ABB RobotStudio station: Solution 4 with position track.rspag

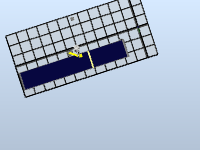
--- station ---
Station Solution4 (saved by RobotStudio 6.8.8148.134)
Controller System1, task T_ROB1: task frame (RAPID world) sits at (5535.63, 748.67, 709.58) mm in the station
Controller System1
  mechanical unit ROB_1: IRB1600_10_145__01, 6 joints, base frame (480.91, -513.23, -359.58) mm, rotated rx 0 ry 0 rz 90 deg
  mechanical unit CNV1: ?, 1 joints, base frame (0, 0, 0) mm
Layout (positions relative to the parent item):
  - bin mover_3 [smart component, from libraries\bin mover.rslib] at (-500, 0, 0) mm
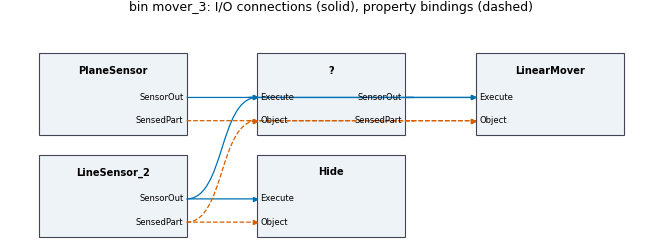
      connections:
        ?.SensorOut -> LinearMover.Execute
        PlaneSensor.SensorOut -> LinearMover.Execute
        ?.SensorOut -> ?.Execute
        LineSensor_2.SensorOut -> ?.Execute
        LineSensor_2.SensorOut -> Hide.Execute
        ?.SensedPart => LinearMover.Object
        PlaneSensor.SensedPart => LinearMover.Object
        ?.SensedPart => ?.Object
        LineSensor_2.SensedPart => ?.Object
        LineSensor_2.SensedPart => Hide.Object
    - LinearMover [smart component, from Components\LinearMover.rslib] at (6663.26, 677.27, 1050.93) mm, rotated rx 180 ry 0 rz 90 deg
        properties: Object=(none); Direction=[0 0 -1]; Speed=8; Reference=Global; ReferenceObject=(none)
    - PlaneSensor [smart component, from Components\PlaneSensor.rslib]
        properties: Origin=[7.419145 0.146999 1.42]; Axis1=[0 0 -1.35]; Axis2=[0 0.4 0]; SensedPart=(none)
      - _sensorPart_ [part, from libraries\bin mover.rslib]
    - LineSensor_2 [smart component, from Components\LineSensor.rslib]
        properties: Start=[7.369145 0.346999 0.008]; End=[7.369145 0.346999 0.123]; Radius=0.09; SensedPart=(none); SensedPoint=[0 0 0]
      - _sensorPart_ [part, from libraries\bin mover.rslib]
    - Hide [smart component, from Components\Hide.rslib]
        properties: Object=(none)
  - bin1_2 [part, from libraries\bin1.rslib] at (6733.74, 347, -12) mm
  - conveyor 1 [part] at (0, -1500, -4460) mm, rotated rx 90 ry 0 rz 90 deg
  - Suction gripper 18cm [smart component] at (6041.96, 965.18, 1386.5) mm, rotated rx 180 ry 0 rz -90 deg
      signals: DI do1
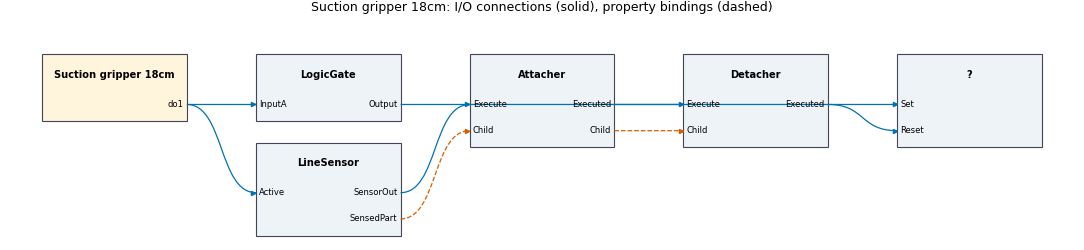
      connections:
        Suction gripper 18cm.do1 -> LogicGate.InputA
        Suction gripper 18cm.do1 -> LineSensor.Active
        LogicGate.Output -> Detacher.Execute
        LineSensor.SensorOut -> Attacher.Execute
        Attacher.Executed -> ?.Set
        Detacher.Executed -> ?.Reset
        LineSensor.SensedPart => Attacher.Child
        Attacher.Child => Detacher.Child
    - Attacher [smart component, from Components\Attacher.rslib]
        properties: Parent=Suction_gripper 18cm; Flange=0; Child=Yellow block; Mount=false; Offset=[0 0 0]; Orientation=[0 0 0]
    - LogicGate [smart component, from Components\LogicGate.rslib]
        properties: Operator=NOT; Delay=0
    - LineSensor [smart component, from Components\LineSensor.rslib] at (7150.29, 306.47, 1168.39) mm, rotated rx 180 ry 0 rz 90 deg
        properties: Start=[-0.30577796087058 -7.14894421240012 1.16938863540814]; End=[-0.305777964813962 -7.14894420825673 1.13938863540814]; Radius=0.09; SensedPart=Yellow block; SensedPoint=[6.72294091796875 0.422247802734375 1.36320727539063]
      - _sensorPart_ [part]
    - Detacher [smart component, from Components\Detacher.rslib]
        properties: Child=Yellow block; KeepPosition=true
  - Suction_gripper 18cm [mechanism, from libraries\Suction_gripper_18cm.rslib] at (6041.96, 965.18, 1471.5) mm, rotated rx 180 ry 0 rz -90 deg
  - IRB1600_10_145__01 [mechanism, from Robots\IRB1600_10_145_G_01.rslib] at (6016.55, 235.44, 350) mm, rotated rx 0 ry 0 rz 90 deg; joint values [-0.0348, -0.0283, 0.0278, 0, 1.5713, -0.0348] (rad or m)
  - 输送链 [conveyor]
    - Conveyor cover [part] at (-300, 0, 14) mm
    - Yellow block [part] at (0, -475.41, 0) mm
    - 传送带对象_37 [conveyorobject] at (9300.11, 748.67, 709.58) mm
      - Yellow block [part] at (-383.96, -1767.23, -1501.67) mm
    - 传送带对象_38 [conveyorobject] at (6600.11, 748.67, 709.58) mm
      - Yellow block [part] at (-344.85, -1769.56, -1503.25) mm
    - 传送带对象_39 [conveyorobject] at (3900.11, 748.67, 709.58) mm
      - Yellow block [part] at (-1067.12, -1221.88, -152.65) mm
  - SmartComponent_1 [smart component]
      signals: DI do_rapid
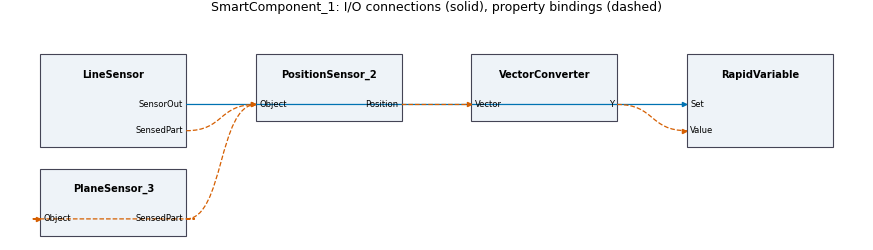
      connections:
        LineSensor.SensorOut -> RapidVariable.Set
        PlaneSensor_3.SensedPart => LinearMover.Object
        PlaneSensor_3.SensedPart => PositionSensor_2.Object
        LineSensor.SensedPart => PositionSensor_2.Object
        PositionSensor_2.Position => VectorConverter.Vector
        VectorConverter.Y => RapidVariable.Value
    - RapidVariable [smart component, from Components\RapidVariable.rslib]
        properties: DataType=num; Controller=System1; Task=T_ROB1; Module=Module1; Variable=y; Value=0.20905832662045
    - PositionSensor_2 [smart component, from Components\PositionSensor.rslib]
        properties: Object=(none); Reference=Object; ReferenceObject=Reference; Position=[-0.750554000259359 0.20905832662045 -0.741395]; Orientation=[0 0 0]
    - LineSensor [smart component, from Components\LineSensor.rslib]
        properties: Start=[5.101063 2.339147 0.72958]; End=[5.101063 0.739147 0.72958]; Radius=0.02; SensedPart=(none); SensedPoint=[0 0 0]
      - _sensorPart_ [part]
    - VectorConverter [smart component, from Components\VectorConverter.rslib]
        properties: X=-0.750554000259359; Y=0.20905832662045; Z=-0.741395; Vector=[-0.750554000259359 0.20905832662045 -0.741395]
  - Reference [part] at (3022.67, -345.33, 752.97) mm
  - Random position [smart component]
      connections:
        PlaneSensor.SensorOut -> Random.Execute
        PlaneSensor.SensorOut -> LinearMover.Execute
        PlaneSensor.SensedPart => LinearMover.Object
        Random.Value => LinearMover.Speed
    - Random [smart component, from Components\Random.rslib]
        properties: Value=0.673263867373236; Min=-0.1; Max=1.2
    - PlaneSensor [smart component, from Components\PlaneSensor.rslib]
        properties: Origin=[4.525795 0.752121 0.710084]; Axis1=[0 0 0.18]; Axis2=[0 1.575 0]; SensedPart=(none)
      - _sensorPart_ [part]
    - LinearMover [smart component, from Components\LinearMover.rslib]
        properties: Object=(none); Direction=[0 0.001 0]; Speed=0.673263867373236; Reference=Global; ReferenceObject=(none)
Attachment: Suction gripper 18cm is attached to Suction_gripper 18cm / Suction gripper 18cm
Attachment: Suction_gripper 18cm is attached to IRB1600_10_145__01 / Link6
Conveyor tracking 连接_2: unit CNV1, TravelOffset=3.7, QueueTrackDistance=0, StartWindowWidth=1.8, SyncSeparation=0, CountsPerMeter=10000
Station logic (signal -> signal, property => property):
  System1.do_attach -> Suction gripper 18cm.do1

--- Backups/System1/RAPID/TASK1/PROGMOD/CalibData.mod ---
MODULE CalibData
	TASK PERS wobjdata wobj_cnv1:=[FALSE,FALSE,"CNV1",[[0,0,0],[1,0,0,0]],[[0,0,0],[1,0,0,0]]];
ENDMODULE

--- Backups/System1/RAPID/TASK1/PROGMOD/Module1.mod ---
MODULE Module1
    VAR num y:=0;
	CONST robtarget Target_10:=[[480.915,236.77,676.92],[0,-0.707106781,0.707106781,0],[0,0,0,0],[9E+09,9E+09,9E+09,9E+09,9E+09,0]];
	CONST robtarget Target_20:=[[29.699626144,355.874016057,111.58001204],[0.000000002,0.707106781,-0.707106781,0.000000007],[0,-1,0,0],[9E+09,9E+09,9E+09,9E+09,9E+09,0]];
	CONST robtarget Target_30:=[[1192.207950487,-330.312717415,676.919992598],[0.000000021,0.707106781,-0.707106781,0.000000022],[-1,-1,-1,0],[9E+09,9E+09,9E+09,9E+09,9E+09,0]];
    PERS tooldata Suction_gripper_18cm:=[TRUE,[[0,0,85],[1,0,0,0]],[1,[0,0,1],[1,0,0,0],0,0,0]];

    PROC main()
        ActUnit CNV1;

        WHILE 2>1 DO

            WaitWObj wobj_cnv1;
            Path_10;
            DropWObj wobj_cnv1;

        ENDWHILE
    ENDPROC
    PROC Path_10()
		MoveL Target_10,vmax,fine,Suction_gripper_18cm\WObj:=wobj0;
		MoveL reltool(Target_20,-y*1000,0,0),vmax,z10,Suction_gripper_18cm\WObj:=wobj_cnv1;
		Set do_attach;
		MoveL Target_30,vmax,fine,Suction_gripper_18cm\WObj:=wobj0;
		Reset do_attach;
		MoveL Target_10,vmax,fine,Suction_gripper_18cm\WObj:=wobj0;

    ENDPROC
ENDMODULE

--- Backups/System1/SYSPAR/EIO.cfg ---
EIO:CFG_1.0:6:1::
#
INDUSTRIAL_NETWORK:

      -Name "RobICI" -Label "RobICI Network"

      -Name "DeviceNet" -Label "DeviceNet Master/Slave Network" -Address "2"
#
ROBICI_DEVICE:

      -Name "CTM1" -TrustLevel "InternalDeviceTrustLevel"\
      -VendorName "ABB Robotics" -ProductName "DSQC2000"\
      -Label "Conveyor Tracking Device 1" -Address "0.0.0.0"
#
DEVICENET_INTERNAL_DEVICE:

      -Name "DN_Internal_Device" -VendorName "ABB Robotics"\
      -ProductName "DeviceNet Internal Slave Device"
#
EIO_SIGNAL:

      -Name "c1Counts" -SignalType "GI" -Device "CTM1"\
      -DeviceMap "Enc1:position"

      -Name "c1CountsPerSec" -SignalType "AI" -Device "CTM1"\
      -DeviceMap "Enc1:velocity"

      -Name "c1TrigVis" -SignalType "DO" -Device "CTM1" -Label "Trig X21 pin 5"\
      -DeviceMap "Digout1:Setpoint"

      -Name "c1TrigAutoMode" -SignalType "DO" -Device "CTM1"\
      -DeviceMap "Cam1:Connect"

      -Name "c1TrigAutoDist" -SignalType "GO" -Device "CTM1"\
      -DeviceMap "Cam1:Interval"

      -Name "c1TrigAutoEncNo" -SignalType "GO" -Device "CTM1"\
      -DeviceMap "Cam1Enc:DeviceNo"

      -Name "c1CntFromEnc" -SignalType "GI" -Device "CTM1"\
      -DeviceMap "Sync1Enc1:Value"

      -Name "c1SoftSync" -SignalType "DO" -Device "CTM1"\
      -DeviceMap "Sync1Enc1:SyncTrig"

      -Name "c1SpeedBandWidth" -SignalType "GI" -Device "CTM1"\
      -DeviceMap "e1_SpeedBandWidth:SetPoint"

      -Name "c1Position" -SignalType "AO" -MaxLog 21474.8 -MaxPhys 1\
      -MaxPhysLimit 1 -MaxBitVal 2147483647 -MinLog -21474.8 -MinPhys -1\
      -MinPhysLimit -1 -MinBitVal -2147483647 -Size 32

      -Name "c1Speed" -SignalType "AO" -MaxLog 21474.8 -MaxPhys 1\
      -MaxPhysLimit 1 -MaxBitVal 2147483647 -MinLog -21474.8 -MinPhys -1\
      -MinPhysLimit -1 -MinBitVal -2147483647 -Size 32

      -Name "c1Connected" -SignalType "DO"

      -Name "c1NullSpeed" -SignalType "DO"

      -Name "c1PassStw" -SignalType "DO"

      -Name "c1NewObjStrobe" -SignalType "DO"

      -Name "c1WaitWObj" -SignalType "DO"

      -Name "c1DropWObj" -SignalType "DO" -Access "ALL"

      -Name "c1Rem1PObj" -SignalType "DO" -Access "All"

      -Name "c1RemAllPObj" -SignalType "DO" -Access "All"

      -Name "c1CntToEncStr" -SignalType "DO"

      -Name "c1PosInJobQ" -SignalType "DO" -Default 1

      -Name "c1ObjectsInQ" -SignalType "GO" -Size 8

      -Name "c1CntToEnc" -SignalType "GO" -Size 32

      -Name "do_attach" -SignalType "DO"

--- Backups/System1/SYSPAR/PROC.cfg ---
PROC:CFG_1.0:6:0::
#
CONVEYOR:

      -name "CNV1" -sensor_type "ICI" -use_sensor "ICI1" -adjustment_speed 850\
      -min_dist -100 -max_dist 20000 -correction_vector_ramp_length 5
#
CONVEYOR_ICI_SENSOR:

      -name "ICI1" -connected_signal "c1Connected" -position_signal "c1Position"\
      -velocity_signal "c1Speed" -position_count_signal "c1Counts"\
      -velocity_count_signal "c1CountsPerSec" -null_speed_signal "c1NullSpeed"\
      -wait_wobj_signal "c1WaitWObj" -drop_wobj_signal "c1DropWObj"\
      -rem_all_pobj_signal "c1RemAllPObj" -rem_one_pobj_signal "c1Rem1PObj"\
      -supervise_max_dist_off  -newobj_strobe "c1NewObjStrobe"\
      -count_to_enc_strobe "c1CntToEncStr" -obj_in_queue_signal "c1ObjectsInQ"\
      -count_from_enc "c1CntFromEnc" -count_to_enc "c1CntToEnc"\
      -StartWinWidth 1.8 -speed_filter_bandwidth "c1SpeedBandWidth"
